//---------------------------------------------------------------------------------------------------------------
//
//  fb_Configuration
//
//  HAUD 2023.04.14
//  - base xml integration
//
//  HAUD 2026.04.10.
//  - now extending a base class
//
//  - cyclic OnChange wrapper for xml data 
//      - Ctrl/State
//        1. INIT
//        2. READ / WRITE
//
//  - read  ST_STATION_PARAMETER on demand
//  - write ST_STATION_PARAMETER on demand
//
//---------------------------------------------------------------------------------------------------------------
// This SOFTWARE is provided as an Example by THE PROVIDER "as is" and "with all faults." THE PROVIDER makes no 
// representations or warranties of any kind concerning the safety, suitability, lack of viruses, inaccuracies, 
// typographical errors, or other harmful components of this SOFTWARE. There are inherent dangers in the use of 
// any software, and you are solely responsible for determining whether this SOFTWARE is compatible with your 
// equipment and other software installed on your equipment. You are also solely responsible for the protection 
// of your equipment and backup of your data, and THE PROVIDER will not be liable for any damages you may suffer 
// in connection with using, modifying, or distributing this SOFTWARE.
//---------------------------------------------------------------------------------------------------------------
FUNCTION_BLOCK fb_Configuration EXTENDS fb_XmlBase
VAR
  _stCtrl               : REFERENCE TO ST_DATA_CTRL;
  _stState              : REFERENCE TO ST_DATA_STATE;

  _stConfiguration      : ST_Configuration;
  _pStationParameter    : POINTER TO ARRAY[1..MAX_STATION] OF ST_STATION_PARAMETER;
END_VAR
VAR CONSTANT
  FILE_ROOT             : STRING := 'CONFIG_XtsTransport_';
  X_PATH                : STRING := '/XtsTransport/config';
END_VAR

//---------------------------------------------------------------------------------------------------------------
//  check pointers from the outside
//---------------------------------------------------------------------------------------------------------------
IF NOT Check() THEN RETURN; END_IF
//---------------------------------------------------------------------------------------------------------------
// always build the internal data pointer
//  - as always: better safe than sorry
//  - leave this bit here, it doesn't cost much and safely addresses the data
//---------------------------------------------------------------------------------------------------------------
_pData                        := ADR    (_stConfiguration);
_nData                        := SIZEOF (_stConfiguration);
_sXpath                       := X_PATH;

// copy to local for debug
_eCmd                         := _stCtrl.Cmd;

// cyclic check for command change
// get state for cmd
IF (_eCmd <> _eCmdOld)
THEN
  // get matching sdtate for Ctrl.Cmd
  _eState                     := Cmd(_eCmd);
  _eCmdOld                    := _eCmd;
END_IF


CASE _eResult
OF
  E_PROGRESS.PROGRESS_INVALID:
    _stState.State            := E_DATA_STATE.NULL;

  E_PROGRESS.PROGRESS_ERROR:
    _stState.State            := _eState + E_PROGRESS.PROGRESS_ERROR;

  E_PROGRESS.PROGRESS_DONE:
    _stState.State            := _eState + E_PROGRESS.PROGRESS_DONE;

ELSE
  // work in progress
  // update progress for extern use
  _stState.State              := _eState + _eResult;

  CASE _eState
  OF
    E_DATA_STATE.INIT:
      _eResult   := _eInit    := CreateFolder(TRUE);

    E_DATA_STATE.READ:
      _eResult                := XmlRead(TRUE);
      IF (_eResult = E_PROGRESS.PROGRESS_DONE)
      THEN
        // copy the single ladies
        memcpy(_pStationParameter, ADR(_stConfiguration.XtsStationParameter), SIZEOF(_stConfiguration.XtsStationParameter));
      END_IF

    E_DATA_STATE.WRITE:
      _eResult                := XmlWrite(TRUE);
  ELSE
      _eResult                := E_PROGRESS.PROGRESS_INVALID;
  END_CASE
END_CASE

METHOD Check : BOOL
//-------------------------------------------------------------------------
IF NOT (__ISVALIDREF(_stCtrl))
THEN
  _eCheck               := E_DATA_CHECK.REFERENCE_CTRL_INVALID;
  RETURN;
END_IF
//-------------------------------------------------------------------------
IF NOT (__ISVALIDREF(_stState))
THEN
  _eCheck               := E_DATA_CHECK.REFERENCE_STATE_INVALID;
  RETURN;
END_IF
//-------------------------------------------------------------------------
IF NOT (_pStationParameter <> 0)
THEN
  _eCheck               := E_DATA_CHECK.POINTER_STATION_PARAMETER_INVALID;
  RETURN;
END_IF
//-------------------------------------------------------------------------
_eCheck                 := E_DATA_CHECK.DONE_CHECK;
Check                   := TRUE;
END_METHOD

METHOD PRIVATE Cmd : E_DATA_STATE
VAR_INPUT
  Ctrl      : E_DATA_CTRL;
END_VAR
VAR_INST
  _eState   : E_DATA_STATE;
END_VAR
IF NOT Check() THEN Cmd   := E_DATA_STATE.NULL;  RETURN; END_IF

CASE Ctrl
OF
  //---------------------------------------------------------------
  E_DATA_CTRL.INIT:
    _sName                := concat(FILE_ROOT, _sIdentity);
    _sName                := concat(_sName, '.xml');
    _sFilePath            := concat(_sDirectoryPath, _sName);

    _eInit                := E_PROGRESS.PROGRESS_INVALID;
    _eResult              := CreateFolder(FALSE);
    _eState               := E_DATA_STATE.INIT;
  //---------------------------------------------------------------
  E_DATA_CTRL.READ:
    _eResult              := XmlRead(FALSE);
    _eState               := E_DATA_STATE.READ;
  //---------------------------------------------------------------
  E_DATA_CTRL.WRITE:
    _stConfiguration.XtsStationParameter  := _pStationParameter^;

    _eResult              := XmlWrite(FALSE);
    _eState               := E_DATA_STATE.WRITE;
ELSE
  //---------------------------------------------------------------
    _eResult              := E_PROGRESS.PROGRESS_INVALID; 
    _eState               := E_DATA_STATE.NO_EXIST;
END_CASE

Cmd                       := _eState;
END_METHOD

PROPERTY Ctrl : REFERENCE to ST_DATA_CTRL
SET
_stCtrl ref= Ctrl;
END_SET
END_PROPERTY

PROPERTY Identity : OTCID
GET
Identity := _XpuIdentity;
END_GET
SET
_XpuIdentity  := Identity;
_sIdentity    := Tc2_Utilities.DWORD_TO_HEXSTR(_XpuIdentity,8,FALSE);
END_SET
END_PROPERTY

PROPERTY State : REFERENCE TO ST_DATA_STATE
SET
_stState ref= State;
END_SET
END_PROPERTY

PROPERTY StationParameter : pointer to ARRAY[1..MAX_STATION] OF ST_STATION_PARAMETER
SET
_pStationParameter := StationParameter;
END_SET
END_PROPERTY

END_FUNCTION_BLOCK

(* stored: Version 1.1.0.1
   POU fb_Configuration: Id {e8c0201e-fc12-4ba0-adbb-972591141a82}, SpecialFunc None
   Folder methods: Id {5561bd3c-d50e-482b-8712-1e34c96de41a}
   Folder properties: Id {987dcc62-838b-4411-ac27-8007621174c9}
   Method Check: Id {59ca6a81-cb86-4c2e-b213-4eff55a05b8b}
   Method Cmd: Id {f52b1230-b416-460e-b3ce-0346aff1e8fc}
   Property Ctrl: Id {9bb8e059-b2ff-46bc-81c8-1c7fc3925274}
   Set Set: Id {7c8785fa-da50-4d0a-ae7f-5cf95124a238}
   Property Identity: Id {3c401dde-7f7c-48f0-975e-4f9eaa179044}
   Get Get: Id {8f79ce27-b32f-41d5-bd58-ce6fcaa82c33}
   Set Set: Id {ab8a305e-3880-4b42-86d1-663fcc255861}
   Property State: Id {706bbe5d-d13c-421d-801c-22265d3341a8}
   Set Set: Id {188ccb9b-962c-422e-8828-5120319fea8b}
   Property StationParameter: Id {bb1dcf6e-ad09-4db8-8b1e-030e6f286194}
   Set Set: Id {1ab52b03-d5a4-416c-9396-6908a14606d1} *)
